{attribute addProperty BoxType "EK1122-0000-0018"}
{attribute addProperty Id "Beckhoff_ATH2xxxsub_EK1100EK1100_179A0949162A_0001_ATH2000_0250_0022A_0001_ATH2000_0250_0022_20236C4E9812.25A_0002_ATH2000_0250_0023A_0002_ATH2000_0250_0023_D700A2ED9812.25A_0003_ATH2000_0250_0024ATH2000_BA5A954865882.25A_0004_ATH2040_0250_0022ATH2040_BA5A954865882.25A_0005_ATH2040_0250_0023ATH2040_BA5A954865882.25A_0006_ATH2040_0250_0024ATH2040_BA5A954865882.25A_0007_ATH2050_0500_0022ATH2050_BA5A954865882.25A_0008_ATH2050_0500_0023ATH2050_BA5A954865882.25A_0009_ATH2050_0500_0024ATH2050_BA5A954865882.25A_0010_ATH2050_0501_0022ATH2050_BA5A954865882.25A_0011_ATH2050_0501_0023ATH2050_BA5A954865882.25A_0012_ATH2050_0501_0024ATH2050_BA5A954865882.25"}
{attribute addProperty CRC "335272960"}
{attribute addProperty SizeInBites "6792"}
{attribute addProperty SizeInBytes "849"}
TYPE Beckhoff_ATH2xxxEK1122_13FBDC00 EXTENDS EK1122_179A0949 :
STRUCT
	{attribute addProperty Name "Beckhoff_ATH2xxxsub_EK1100"}
	Beckhoff_ATH2xxxsub_EK1100 : EK1100_179A0949;
	{attribute addProperty Name "A_0001_ATH2000_0250_0022"}
	A_0001_ATH2000_0250_0022 : A_0001_ATH2000_0250_0022_20236C4E;
	{attribute addProperty Name "A_0002_ATH2000_0250_0023"}
	A_0002_ATH2000_0250_0023 : A_0002_ATH2000_0250_0023_D700A2ED;
	{attribute addProperty Name "A_0003_ATH2000_0250_0024"}
	A_0003_ATH2000_0250_0024 : ATH2000_BA5A9548;
	{attribute addProperty Name "A_0004_ATH2040_0250_0022"}
	A_0004_ATH2040_0250_0022 : ATH2040_BA5A9548;
	{attribute addProperty Name "A_0005_ATH2040_0250_0023"}
	A_0005_ATH2040_0250_0023 : ATH2040_BA5A9548;
	{attribute addProperty Name "A_0006_ATH2040_0250_0024"}
	A_0006_ATH2040_0250_0024 : ATH2040_BA5A9548;
	{attribute addProperty Name "A_0007_ATH2050_0500_0022"}
	A_0007_ATH2050_0500_0022 : ATH2050_BA5A9548;
	{attribute addProperty Name "A_0008_ATH2050_0500_0023"}
	A_0008_ATH2050_0500_0023 : ATH2050_BA5A9548;
	{attribute addProperty Name "A_0009_ATH2050_0500_0024"}
	A_0009_ATH2050_0500_0024 : ATH2050_BA5A9548;
	{attribute addProperty Name "A_0010_ATH2050_0501_0022"}
	A_0010_ATH2050_0501_0022 : ATH2050_BA5A9548;
	{attribute addProperty Name "A_0011_ATH2050_0501_0023"}
	A_0011_ATH2050_0501_0023 : ATH2050_BA5A9548;
	{attribute addProperty Name "A_0012_ATH2050_0501_0024"}
	A_0012_ATH2050_0501_0024 : ATH2050_BA5A9548;
END_STRUCT
END_TYPE

(* stored: Version 1.2.0.0, ProductVersion 3.1.4024.9
   DUT Beckhoff_ATH2xxxEK1122_13FBDC00: Id {15325b28-21b1-4737-ac4a-1f602a63b0e7} *)
